TYPE Status :
STRUCT
	Enable:BOOL;					//使能状态
	Velocity:LREAL;					//速度状态
	Position:LREAL;					//位置状态
END_STRUCT
END_TYPE

(* stored: Version 1.1.0.1, ProductVersion 3.1.4022.10
   DUT Status: Id {e251c0c9-1caa-44a9-8432-5824f0b26c96} *)
